FUNCTION_BLOCK PUBLIC ABSTRACT TcoUrRoboticsTask EXTENDS TcoCore.TcoTask 
VAR_IN_OUT
    inoConfig 	: TcoUrRobotics_Config_v_1_x_x;
	inoControl 	: TcoUrRobotics_Control_v_1_x_x;
	inoStatus 	: TcoUrRobotics_Status_v_1_x_x;	
END_VAR
VAR
	_errorMessage:TcoCore.TcoMessenger(THIS^);
    {attribute 'hide'} 
	_progress : INT := 0;
    {attribute 'hide'} 
	_infoTimer :  TON;
    {attribute 'hide'} 
	_errorTimer :  TON;
	{attribute 'hide'} 
	_timer :  TON;
    {attribute 'hide'} 
	_varInfo : __SYSTEM.VAR_INFO;
    {attribute 'hide'} 
	_sb : TcoCore.StringBuilder;
	{attribute 'hide'}
	_blink:TcoUtilities.TcoBlinker(THIS^);
END_VAR

METHOD CallTimers
VAR_INPUT
	inValue : BOOL;
END_VAR
IF  __ISVALIDREF(inoConfig) AND THIS^.inoConfig.ErrorTime <> T#0S OR NOT inValue THEN  
_errorTimer(IN := inValue, PT := THIS^.inoConfig.ErrorTime);
END_IF;
IF  __ISVALIDREF(inoConfig) AND THIS^.inoConfig.InfoTime <>T#0S OR NOT inValue THEN  
_infoTimer(IN := inValue, PT := THIS^.inoConfig.InfoTime);
END_IF;
END_METHOD

(*~
	<docu>
		<summary>
			Restores this instance to the Ready state. Can be called explicitly or from within one of the restore mechanisms.
			<para>
				See also <see cref="PlcDocu.TcoCore.TcoTask.AutoRestorable()"/>
			</para>
		</summary>			
	</docu>	
~*)
METHOD Restore : ITcoRestorable
SUPER^.Restore();
_progress := 0;
_timer(In:=FALSE);
CallTimers(FALSE);
Messenger.UnPin();
_errorMessage.UnPin();
END_METHOD

END_FUNCTION_BLOCK

(* stored: Version 1.1.0.1, ProductVersion 3.1.4024.12
   POU TcoUrRoboticsTask: Id {e690c3a2-6f40-0358-3fb9-61b724057750}, SpecialFunc None
   Method CallTimers: Id {b922e381-15be-0484-1dda-96171d80bbd6}
   Method Restore: Id {fd91723e-954c-0524-3405-f97f744cd643} *)
